Staubli VAL3: _DetectIOEdge.pgx

program _DetectIOEdge(bool x_bInput (dimensions=1), bool& x_bMemoState[] (dimensions=1), bool& x_bRisingEdge[] (dimensions=1))
begin
  // ABSTRACT
  // This program checks if a transition from TRUE to FALSE
  // occured on the boolean expression passed as parameter. This routine is usually
  // used to detect rising/falling edge on digital inputs.
  //
  // Input Param
  //x_bInput    : Boolean expression to evaluate
  //
  // Output Param
  //x_bMemoState    : Memory of the boolean expression value
  //x_bEdgeDetected : True if transition from TRUE to FALSE occured
  //
  // Comments : Ladder diagram
  //Raising Edge
  //|---[x_bInput]---[/x_bMemoState]---(x_bRaisEdge)--|
  //
  //|---[x_bInput]--------------------(x_bMemoState)--|
  //
  x_bRisingEdge=(x_bInput) and !x_bMemoState
  //x_bFallEdge=!x_bInput and (x_bMemoState)
  x_bMemoState=(x_bInput)
end
